// TIA Portal V17 export
// export: Created 2021-12-03T08:12:56.7873031Z, ExportSetting WithDefaults, DisplayName Totally Integrated Automation Portal, DisplayVersion V17, DisplayName TIA Portal Openness, DisplayVersion V17, DisplayName TIA Portal Version Control Interface, DisplayVersion V17, DisplayName STEP 7 Professional, DisplayVersion V17, DisplayName STEP 7 Safety, DisplayVersion V17, DisplayName WinCC Advanced, DisplayVersion V17
ORGANIZATION_BLOCK "Main"   // OB1, FBD, ProgramCycle
TITLE = "Main Program Sweep (Cycle)"
VERSION : 0.1
// stored: IsIECCheckEnabled false
   VAR_TEMP
      OB1_EV_CLASS : Byte;   // Bits 0-3 = 1 (Coming event), Bits 4-7 = 1 (Event class 1)
      OB1_SCAN_1 : Byte;   // 1 (Cold restart scan 1 of OB 1), 3 (Scan 2-n of OB 1)
      OB1_PRIORITY : Byte;   // Priority of OB Execution
      OB1_OB_NUMBR : Byte;   // 1 (Organization block 1, OB1)
      OB1_RESERVED_1 : Byte;   // Reserved for system
      OB1_RESERVED_2 : Byte;   // Reserved for system
      OB1_PREV_CYCLE : Int;   // Cycle time of previous OB1 scan (milliseconds)
      OB1_MIN_CYCLE : Int;   // Minimum cycle time of OB1 (milliseconds)
      OB1_MAX_CYCLE : Int;   // Maximum cycle time of OB1 (milliseconds)
      OB1_DATE_TIME : Date_And_Time;   // Date and time OB1 started
   END_VAR
BEGIN

REGION Network 1: Чтение входов
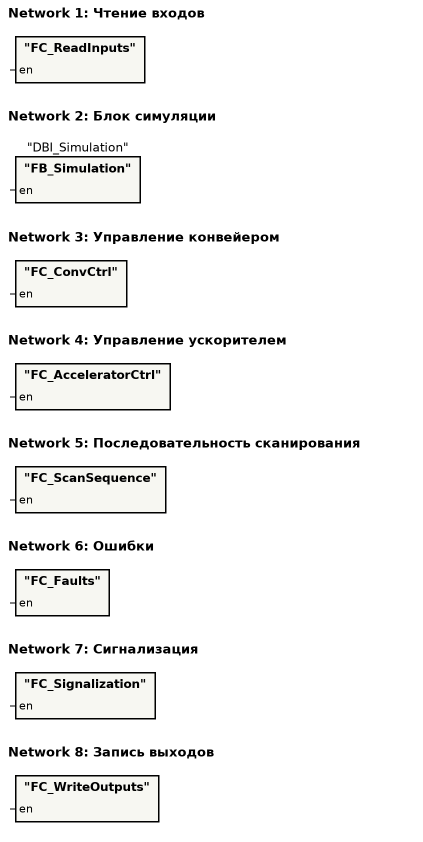
   "FC_ReadInputs"();
END_REGION

REGION Network 2: Блок симуляции
   "DBI_Simulation"();   // "FB_Simulation"
END_REGION

REGION Network 3: Управление конвейером
   "FC_ConvCtrl"();
END_REGION

REGION Network 4: Управление ускорителем
   "FC_AcceleratorCtrl"();
END_REGION

REGION Network 5: Последовательность сканирования
   "FC_ScanSequence"();
END_REGION

REGION Network 6: Ошибки
   "FC_Faults"();
END_REGION

REGION Network 7: Сигнализация
   "FC_Signalization"();
END_REGION

REGION Network 8: Запись выходов
   "FC_WriteOutputs"();
END_REGION
END_ORGANIZATION_BLOCK
